(* PLC project 117_1_V0.5.project, CODESYS CODESYS V3.5 SP17 Patch 3 *)
(* stored: creationDateTime 1970-01-01T00:00:00, modificationDateTime 2026-03-26T18:14:32.4070562 *)

FUNCTION_BLOCK SM3ServoDriver
  VAR_INPUT
    TimeManager : REFERENCE TO TimeManager;
  END_VAR
  VAR
    _CheckAxisCommuniction : SMC_CheckAxisCommunication;  (* Проверка связи с драйвером *)
    _CheckPowerStatus : MC_ReadBoolParameter;  (* Прверка питания драйвера *)
    _pNum : UINT;
    _powerStatusValue : ARRAY[0..1] OF BOOL;
    _Power : MC_Power;  (* Управление питанием драйвера *)
    _powerSteps : UINT;
    _Jogging : MC_Jog;  (* Ручной режим *)
    _FollowVelocity : SMC_FollowVelocity;  (* Режим управления скоростью *)
    _Reset_Errors : MC_Reset;  (* Сброс аварий *)
    _reset_Enable : BOOL;
    _bErrors : ARRAY[communication..(lastIndex - 1)] OF BOOL;  (* Дата и время для логов Сбор ошобок в слово *)
    _wAxisErrors : BYTE;
    _ErrorsFlag : BOOL;
    _eAxisErrorsID : ARRAY[communication..(lastIndex - 1)] OF SMC_ERROR;  (* Данные для флагов ошибок и записи в лог *)
    _sComments : ARRAY[communication..(lastIndex - 1)] OF STRING(40);
    _trErrorsTrigs : ARRAY[communication..(lastIndex - 1)] OF R_TRIG;
    _axisErrorsLog : ARRAY[0..9] OF STRING(100);  (* Лог *)
    _logSize : UINT;
    _errorIndex : ERROR_INDEX;
  END_VAR
  VAR CONSTANT
    dPowerParameter : ARRAY[0..1] OF DINT := [1015, 1016];
  END_VAR

            // Проверка связи
_CheckAxisCommuniction(
	Axis	:= SM_Drive_GenericDSP402,
	bEnable := TRUE);

//Проверка наличия питания
FOR _pNum := 0 TO 1 DO
	_CheckPowerStatus(
		Axis			:= SM_Drive_GenericDSP402,
		Enable			:= TRUE,
		ParameterNumber	:= dPowerParameter[_pNum],
		Value			=> _powerStatusValue[_pNum]); 
END_FOR

// Питание драйвера
_Power(Axis	:= SM_Drive_GenericDSP402);

// Ручное управление дравером
_Jogging(Axis := SM_Drive_GenericDSP402); 

//Режим управления скоростью
_FollowVelocity(Axis := SM_Drive_GenericDSP402);

// Сброс ошибок
_Reset_Errors(Axis:= SM_Drive_GenericDSP402, Execute:= _reset_Enable); 

// // Запись флагов ошибок ФБ в массив
// _bErrors[communication]	 := _CheckAxisCommuniction.bError;
// _bErrors[power]			 := _Power.Error;
// _bErrors[jogging]		 := _Jogging.Error;
// _bErrors[follow]		 := _FollowVelocity.bError;
// _bErrors[reset]			 := _Reset_Errors.Error;

// Запись ошибок
FOR _errorIndex := communication TO lastIndex - 1 DO
	// Триггеры ошибок для записи в лог	
	_trErrorsTrigs[_errorIndex](CLK := _bErrors[_errorIndex]);
	
	// 	Формирование слова ошибок
    IF _bErrors[_errorIndex] THEN
        _wAxisErrors := _wAxisErrors OR SHL(BYTE#1, _errorIndex);
	ELSE
		_wAxisErrors := _wAxisErrors AND NOT SHL(BYTE#1, _errorIndex);
    END_IF
	
END_FOR

// Идентификаторы ошибок
_eAxisErrorsID	[communication]	:= _CheckAxisCommuniction.eErrorID;
_eAxisErrorsID	[power]			:= _Power.ErrorID;
_eAxisErrorsID	[jogging]		:= _Jogging.ErrorID;
_eAxisErrorsID	[follow]		:= _FollowVelocity.iErrorID;
_eAxisErrorsID	[reset]			:= _Reset_Errors.ErrorID;

//Коментарии к ошибкам
_sComments		[communication] := 'Ошибка при диагностике связи';
_sComments		[power]			:= 'Ошибка при включении питания драйвера';
_sComments		[jogging]		:= 'Ошибка при ручном управлении';
_sComments		[follow]		:= 'Ошибка при управлении скоростью';
_sComments		[reset]			:= 'Ошибка при сбросе ошибок';

// Метод для записи ошибки в лог
FOR _errorIndex := communication TO lastIndex - 1 DO
_error_handler(
	bError		:= _trErrorsTrigs[_errorIndex].Q,
	arrIndex	:= _errorIndex,
	eErrorID	:= _eAxisErrorsID[_errorIndex],
	sComment	:= _sComments[_errorIndex]
);	
END_FOR

_ErrorsFlag	:= _wAxisErrors > 0;





          

METHOD start_backward_jogging : BOOL
  VAR_INPUT
    velocity : LREAL := 0;
    acceleration : LREAL := 0;
    deceleration : LREAL := 0;
    jerk : LREAL := 0;
  END_VAR
                  _Jogging.JogForward		:= FALSE; 
_Jogging.JogBackward	:= TRUE; 
_Jogging.Velocity		:= velocity; 
_Jogging.Acceleration	:= acceleration; 
_Jogging.Deceleration	:= deceleration; 
_Jogging.Jerk			:= jerk; 

start_backward_jogging := _Jogging.Busy;
                
END_METHOD
END_FUNCTION_BLOCK
